{attribute 'GeneratedUsingTerminal: AT2000-0233-0022'}
{attribute addProperty BoxType "AT2000-0233-0022"}
{attribute addProperty Description "AT2000-0233 Motor module 233 mm, 48V"}
{attribute addProperty Physics "YKY"}
{attribute addProperty Id "CC_Inputs_14_ChAT %I*CC_Inputs_14_Ch_F1B7955430CC_Outputs_14_ChAT %Q*CC_Outputs_14_Ch_4596551130WcStateAT %I*WcState_9091E0EB2InfoDataAT %I*InfoData_BEF6B88E18"}
{attribute addProperty CRC "403295535"}
{attribute addProperty Size "80"}
TYPE AT2000_1809CD2F EXTENDS EtcSlaveBoxBase_77A0E4A7 :
STRUCT
	{attribute addProperty Name "CC_Inputs_14_Ch"}
	CC_Inputs_14_Ch : CC_Inputs_14_Ch_F1B79554;
	{attribute addProperty Name "CC_Outputs_14_Ch"}
	CC_Outputs_14_Ch : CC_Outputs_14_Ch_45965511;
	{attribute addProperty Name "WcState"}
	WcState : WcState_9091E0EB;
	{attribute addProperty Name "InfoData"}
	InfoData : InfoData_BEF6B88E;
END_STRUCT
END_TYPE

(* stored: Version 1.2.0.0, ProductVersion 3.1.4024.9
   DUT AT2000_1809CD2F: Id {6083dbee-bdfa-4bba-80fa-2db6bb113f73} *)
